{attribute 'qualified_only'}


//{attribute 'strict'}



  {attribute 'to_string'}
 TYPE E_MachineState :


(
_ABORTING := 0,
 _ABORTED,
 _CLEARING,
 _STOPPED,
 _RESETING,
 _IDLE,
 _STARTING,
 _EXECUTE,
 _COMPLETE


);


END_TYPE

(* stored: Version 1.1.0.1, ProductVersion 3.1.4024.12
   DUT E_MachineState: Id {c344b96f-96e1-4007-ae2b-bcf79c16f4cd} *)
